{attribute 'Tc2GvlVarNames'}
VAR_CONFIG
END_VAR

(* stored: Version 1.1.0.1, ProductVersion 3.1.4024.12
   GVL Variable_Configuration: Id {d5bcb56a-77d6-4fcb-b94b-21bcb6d63a3f} *)
